(*
============================================================
ST_MQTT_Command
============================================================
PURPOSE
  JSON-deserialized incoming MQTT command payload.
  FB_MqttManager parses received JSON into this struct.

EXPECTED JSON FORMAT (publish to irrigation/command):
  {
    "Valve1": 50,
    "Valve2": 25,
    "Valve3": 75
  }

  Valve setpoints are in percent (0–100).
  Omitting a field leaves its current value unchanged.

NOTES
  • {attribute 'TcJsonObject'} enables Beckhoff JSON auto-parse.
  • DINT used for setpoints to avoid floating-point JSON quirks;
    values are clamped to 0–100 before use.
============================================================
*)
{attribute 'TcJsonObject' := ''}
TYPE ST_MQTT_Command :
STRUCT
    (* ── Setpoints (0–100 %) ────────────────────────────────── *)
    Valve1          : DINT;     (* Desired position valve 1, 0–100 % *)
    Valve2          : DINT;     (* Desired position valve 2, 0–100 % *)
    Valve3          : DINT;     (* Desired position valve 3, 0–100 % *)
END_STRUCT
END_TYPE

(* stored: Version 1.1.0.1, ProductVersion 3.1.4026.18
   DUT ST_MQTT_Command: Id {6408835c-1577-4fae-afd9-8d68de3755d2} *)
